# EPICS substitutions: iocBoot/ioc13bmd/ipUnidig.substitutions
file "$(IPUNIDIG)/db/IpUnidigLi.db"
{
pattern
{P,       R,          PORT,       SCAN}
{13BMD:,  Unidig1Li,  Unidig1, "I/O Intr"}
{13BMD:,  Unidig2Li,  Unidig2, "I/O Intr"}
}

file "$(IPUNIDIG)/db/IpUnidigBi.db"
{
pattern
{P,       R,          PORT,    MASK,        SCAN}
{13BMD:, Unidig1Bi0,  Unidig1, 0x000001, "I/O Intr"}
{13BMD:, Unidig1Bi1,  Unidig1, 0x000002, "I/O Intr"}
{13BMD:, Unidig1Bi2,  Unidig1, 0x000004, "1 second"}
{13BMD:, Unidig1Bi3,  Unidig1, 0x000008, "I/O Intr"}
{13BMD:, Unidig1Bi4,  Unidig1, 0x000010, "I/O Intr"}
{13BMD:, Unidig1Bi5,  Unidig1, 0x000020, "I/O Intr"}
{13BMD:, Unidig1Bi6,  Unidig1, 0x000040, "I/O Intr"}
{13BMD:, Unidig1Bi7,  Unidig1, 0x000080, "I/O Intr"}
{13BMD:, Unidig1Bi8,  Unidig1, 0x000100, "I/O Intr"}
{13BMD:, Unidig1Bi9,  Unidig1, 0x000200, "I/O Intr"}
{13BMD:, Unidig1Bi10, Unidig1, 0x000400, "I/O Intr"}
{13BMD:, Unidig1Bi11, Unidig1, 0x000800, "I/O Intr"}
{13BMD:, Unidig1Bi12, Unidig1, 0x001000, "I/O Intr"}
{13BMD:, Unidig1Bi13, Unidig1, 0x002000, "I/O Intr"}
{13BMD:, Unidig1Bi14, Unidig1, 0x004000, "I/O Intr"}
{13BMD:, Unidig1Bi15, Unidig1, 0x008000, "I/O Intr"}
{13BMD:, Unidig1Bi16, Unidig1, 0x010000, "I/O Intr"}
{13BMD:, Unidig1Bi17, Unidig1, 0x020000, "I/O Intr"}
{13BMD:, Unidig1Bi18, Unidig1, 0x040000, "I/O Intr"}
{13BMD:, Unidig1Bi19, Unidig1, 0x080000, "I/O Intr"}
{13BMD:, Unidig1Bi20, Unidig1, 0x100000, "I/O Intr"}
{13BMD:, Unidig1Bi21, Unidig1, 0x200000, "I/O Intr"}
{13BMD:, Unidig1Bi22, Unidig1, 0x400000, "I/O Intr"}
{13BMD:, Unidig1Bi23, Unidig1, 0x800000, "I/O Intr"}
{13BMD:, Unidig2Bi0,  Unidig2, 0x000001, "I/O Intr"}
{13BMD:, Unidig2Bi1,  Unidig2, 0x000002, "I/O Intr"}
{13BMD:, Unidig2Bi2,  Unidig2, 0x000004, "1 second"}
{13BMD:, Unidig2Bi3,  Unidig2, 0x000008, "I/O Intr"}
{13BMD:, Unidig2Bi4,  Unidig2, 0x000010, "I/O Intr"}
{13BMD:, Unidig2Bi5,  Unidig2, 0x000020, "I/O Intr"}
{13BMD:, Unidig2Bi6,  Unidig2, 0x000040, "I/O Intr"}
{13BMD:, Unidig2Bi7,  Unidig2, 0x000080, "I/O Intr"}
{13BMD:, Unidig2Bi8,  Unidig2, 0x000100, "I/O Intr"}
{13BMD:, Unidig2Bi9,  Unidig2, 0x000200, "I/O Intr"}
{13BMD:, Unidig2Bi10, Unidig2, 0x000400, "I/O Intr"}
{13BMD:, Unidig2Bi11, Unidig2, 0x000800, "I/O Intr"}
{13BMD:, Unidig2Bi12, Unidig2, 0x001000, "I/O Intr"}
{13BMD:, Unidig2Bi13, Unidig2, 0x002000, "I/O Intr"}
{13BMD:, Unidig2Bi14, Unidig2, 0x004000, "I/O Intr"}
{13BMD:, Unidig2Bi15, Unidig2, 0x008000, "I/O Intr"}
{13BMD:, Unidig2Bi16, Unidig2, 0x010000, "I/O Intr"}
{13BMD:, Unidig2Bi17, Unidig2, 0x020000, "I/O Intr"}
{13BMD:, Unidig2Bi18, Unidig2, 0x040000, "I/O Intr"}
{13BMD:, Unidig2Bi19, Unidig2, 0x080000, "I/O Intr"}
{13BMD:, Unidig2Bi20, Unidig2, 0x100000, "I/O Intr"}
{13BMD:, Unidig2Bi21, Unidig2, 0x200000, "I/O Intr"}
{13BMD:, Unidig2Bi22, Unidig2, 0x400000, "I/O Intr"}
{13BMD:, Unidig2Bi23, Unidig2, 0x800000, "I/O Intr"}
}

file "$(IPUNIDIG)/db/IpUnidigBo.db"
{
pattern
{P,       R,        PORT,    MASK}
{13BMD:, Unidig1Bo0,  Unidig1, 0x000001}
{13BMD:, Unidig1Bo1,  Unidig1, 0x000002}
{13BMD:, Unidig1Bo2,  Unidig1, 0x000004}
{13BMD:, Unidig1Bo3,  Unidig1, 0x000008}
{13BMD:, Unidig1Bo4,  Unidig1, 0x000010}
{13BMD:, Unidig1Bo5,  Unidig1, 0x000020}
{13BMD:, Unidig1Bo6,  Unidig1, 0x000040}
{13BMD:, Unidig1Bo7,  Unidig1, 0x000080}
{13BMD:, Unidig1Bo8,  Unidig1, 0x000100}
{13BMD:, Unidig1Bo9,  Unidig1, 0x000200}
{13BMD:, Unidig1Bo10, Unidig1, 0x000400}
{13BMD:, Unidig1Bo11, Unidig1, 0x000800}
{13BMD:, Unidig1Bo12, Unidig1, 0x001000}
{13BMD:, Unidig1Bo13, Unidig1, 0x002000}
{13BMD:, Unidig1Bo14, Unidig1, 0x004000}
{13BMD:, Unidig1Bo15, Unidig1, 0x008000}
{13BMD:, Unidig1Bo16, Unidig1, 0x010000}
{13BMD:, Unidig1Bo17, Unidig1, 0x020000}
{13BMD:, Unidig1Bo18, Unidig1, 0x040000}
{13BMD:, Unidig1Bo19, Unidig1, 0x080000}
{13BMD:, Unidig1Bo20, Unidig1, 0x100000}
{13BMD:, Unidig1Bo21, Unidig1, 0x200000}
{13BMD:, Unidig1Bo22, Unidig1, 0x400000}
{13BMD:, Unidig1Bo23, Unidig1, 0x800000}
{13BMD:, Unidig2Bo0,  Unidig2, 0x000001}
{13BMD:, Unidig2Bo1,  Unidig2, 0x000002}
{13BMD:, Unidig2Bo2,  Unidig2, 0x000004}
{13BMD:, Unidig2Bo3,  Unidig2, 0x000008}
{13BMD:, Unidig2Bo4,  Unidig2, 0x000010}
{13BMD:, Unidig2Bo5,  Unidig2, 0x000020}
{13BMD:, Unidig2Bo6,  Unidig2, 0x000040}
{13BMD:, Unidig2Bo7,  Unidig2, 0x000080}
{13BMD:, Unidig2Bo8,  Unidig2, 0x000100}
{13BMD:, Unidig2Bo9,  Unidig2, 0x000200}
{13BMD:, Unidig2Bo10, Unidig2, 0x000400}
{13BMD:, Unidig2Bo11, Unidig2, 0x000800}
{13BMD:, Unidig2Bo12, Unidig2, 0x001000}
{13BMD:, Unidig2Bo13, Unidig2, 0x002000}
{13BMD:, Unidig2Bo14, Unidig2, 0x004000}
{13BMD:, Unidig2Bo15, Unidig2, 0x008000}
{13BMD:, Unidig2Bo16, Unidig2, 0x010000}
{13BMD:, Unidig2Bo17, Unidig2, 0x020000}
{13BMD:, Unidig2Bo18, Unidig2, 0x040000}
{13BMD:, Unidig2Bo19, Unidig2, 0x080000}
{13BMD:, Unidig2Bo20, Unidig2, 0x100000}
{13BMD:, Unidig2Bo21, Unidig2, 0x200000}
{13BMD:, Unidig2Bo22, Unidig2, 0x400000}
{13BMD:, Unidig2Bo23, Unidig2, 0x800000}
}

file "$(IPUNIDIG)/db/IpUnidigLo.db"
{
pattern
{P,       R,          PORT}
{13BMD:,  Unidig1Lo,  Unidig1}
{13BMD:,  Unidig2Lo,  Unidig2}
}
